FUNCTION F_CalcBCC : BYTE
VAR_INPUT 
	sCore : STRING(160); (* STX..ETX를 포함한 코어 문자열 *) 
END_VAR
VAR 
	i:INT; 
	b:BYTE; 
	sum:UDINT; 
	stxSeen:BOOL; 
END_VAR

sum:=0; 
stxSeen:=FALSE;

FOR i:=1 TO LEN(sCore) DO
	b := TO_BYTE(sCore[i]);
	IF NOT stxSeen THEN
		IF b = GVL_CONSTANT.cSTX THEN 
			stxSeen:=TRUE; 
		END_IF
	ELSE
		IF b = GVL_CONSTANT.cETX THEN 
			EXIT; 
		END_IF
			sum := sum + b;
	END_IF
END_FOR
F_CalcBCC := TO_BYTE(sum MOD 128);

END_FUNCTION

(* stored: Version 1.1.0.1, ProductVersion 3.1.4024.15
   POU F_CalcBCC: Id {1b07d96f-6ebe-4d26-826e-f8bac4362544}, SpecialFunc None *)
